FUNCTION_BLOCK WastewaterControl
VAR_INPUT
    InFlow : REAL; // 进水量(单位：m³/h)
    OutFlow : REAL; // 出水量(单位：m³/h)
    pH : REAL; // 污水pH值
    TankLvl : REAL; // 水箱液位(单位：%)
END_VAR
VAR_OUTPUT
    Pump1 : BOOL; // 泵1控制信号
    Pump2 : BOOL; // 泵2控制信号
    Valve1 : BOOL; // 阀门1控制信号
    Valve2 : BOOL; // 阀门2控制信号
END_VAR
VAR
    // 过程变量常量定义(便于集中管理和修改)
    CONST
        // 输入变量边界范围
        MIN_FLOW : REAL := 0.0; // 流量最小值(单位：m³/h)
        MAX_FLOW : REAL := 1000.0; // 流量最大值(单位：m³/h)
        MIN_PH : REAL := 0.0; // pH最小值
        MAX_PH : REAL := 14.0; // pH最大值
        MIN_TANK_LVL : REAL := 0.0; // 水箱液位最小值(单位：%)
        MAX_TANK_LVL : REAL := 100.0; // 水箱液位最大值(单位：%)
        
        // 控制阈值常量
        LOW_IN_FLOW : REAL := 100.0; // 进水量低阈值(单位：m³/h)
        HIGH_OUT_FLOW : REAL := 90.0; // 出水量高阈值(单位：m³/h)
        DESIRED_PH : REAL := 7.0; // 目标pH值
        HIGH_TANK_LVL : REAL := 80.0; // 水箱液位高阈值(单位：%)
    END_CONST
    
    // 内部处理变量
    FilteredInFlow : REAL; // 过滤后的进水量(单位：m³/h)
    FilteredOutFlow : REAL; // 过滤后的出水量(单位：m³/h)
    FilteredPH : REAL; // 过滤后的pH值
    FilteredTankLvl : REAL; // 过滤后的水箱液位(单位：%)
END_VAR


// 输入变量边界条件处理
FilteredInFlow := LIMIT(MIN_FLOW, InFlow, MAX_FLOW);
FilteredOutFlow := LIMIT(MIN_FLOW, OutFlow, MAX_FLOW);
FilteredPH := LIMIT(MIN_PH, pH, MAX_PH);
FilteredTankLvl := LIMIT(MIN_TANK_LVL, TankLvl, MAX_TANK_LVL);

// 控制逻辑实现
Pump1 := (FilteredInFlow < LOW_IN_FLOW);
Pump2 := (FilteredOutFlow > HIGH_OUT_FLOW);
Valve1 := (FilteredPH < DESIRED_PH);
Valve2 := (FilteredTankLvl > HIGH_TANK_LVL);

// 形式化属性验证断言
ASSERT(
    (FilteredInFlow >= LOW_IN_FLOW) OR Pump1,
    'Assertion failed: InFlow >= 100.0 OR Pump1 = TRUE'
);

ASSERT(
    (FilteredOutFlow <= HIGH_OUT_FLOW) OR Pump2,
    'Assertion failed: OutFlow <= 90.0 OR Pump2 = TRUE'
);

ASSERT(
    (FilteredPH >= DESIRED_PH) OR Valve1,
    'Assertion failed: pH >= 7.0 OR Valve1 = TRUE'
);

ASSERT(
    (FilteredTankLvl <= HIGH_TANK_LVL) OR Valve2,
    'Assertion failed: TankLvl <= 80.0 OR Valve2 = TRUE'
);

END_FUNCTION_BLOCK
